// TIA Portal V20 export
VAR_GLOBAL   // PLC tag table "2.Salida Digital"
   Output_1 AT %Q0.0 : Bool;
   Output_2 AT %Q0.1 : Bool;
   Output_3 AT %Q0.2 : Bool;
   Output_4 AT %Q0.3 : Bool;
   Output_5 AT %Q0.4 : Bool;
   Output_6 AT %Q0.5 : Bool;
   Output_7 AT %Q0.6 : Bool;
   Output_8 AT %Q0.7 : Bool;
   Output_9 AT %Q1.0 : Bool;
   Output_10 AT %Q1.1 : Bool;
   Output_11 AT %Q1.2 : Bool;
   Output_12 AT %Q1.3 : Bool;
   Output_13 AT %Q1.4 : Bool;
   Output_14 AT %Q1.5 : Bool;
   Output_15 AT %Q1.6 : Bool;
   Output_16 AT %Q1.7 : Bool;
END_VAR
